FUNCTION_BLOCK E_MERGE (* Merge (OR) of two input events *)
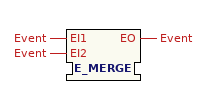
  EVENT_INPUT
    EI1; (* First input event *)
    EI2; (* Second input event *)
  END_EVENT
  EVENT_OUTPUT
    EO; (* Output Event *)
  END_EVENT
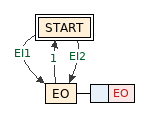
  EC_STATES
    START; (* Initial State *)
    EO : -> EO; (* Issue EO Event *)
  END_STATES
  EC_TRANSITIONS
    EO TO START := 1;
    START TO EO := EI1;
    START TO EO := EI2;
  END_TRANSITIONS
END_FUNCTION_BLOCK
